// Mitsubishi GX Works2 project: 1   PLC: Q03UDV

PROGRAM P1
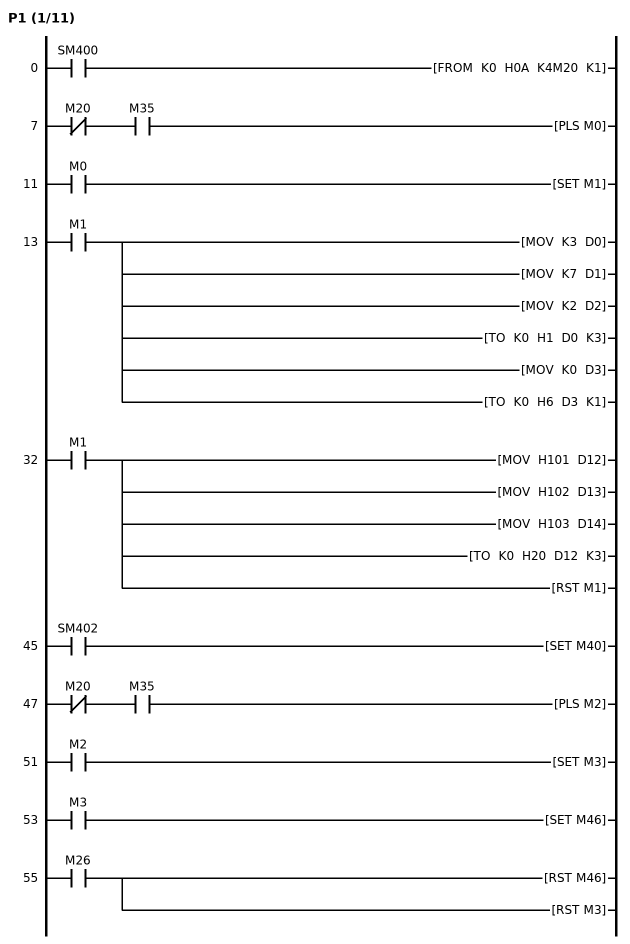
0     LD      SM400
      FROM    K0 H0A K4M20 K1
7     LDI     M20
      AND     M35
      PLS     M0
11    LD      M0
      SET     M1
13    LD      M1
      MOV     K3 D0
      MOV     K7 D1
      MOV     K2 D2
      TO      K0 H1 D0 K3
      MOV     K0 D3
      TO      K0 H6 D3 K1
32    LD      M1
      MOV     H101 D12
      MOV     H102 D13
      MOV     H103 D14
      TO      K0 H20 D12 K3
      RST     M1
45    LD      SM402
      SET     M40
47    LDI     M20
      AND     M35
      PLS     M2
51    LD      M2
      SET     M3
53    LD      M3
      SET     M46
55    LD      M26
      RST     M46
      RST     M3
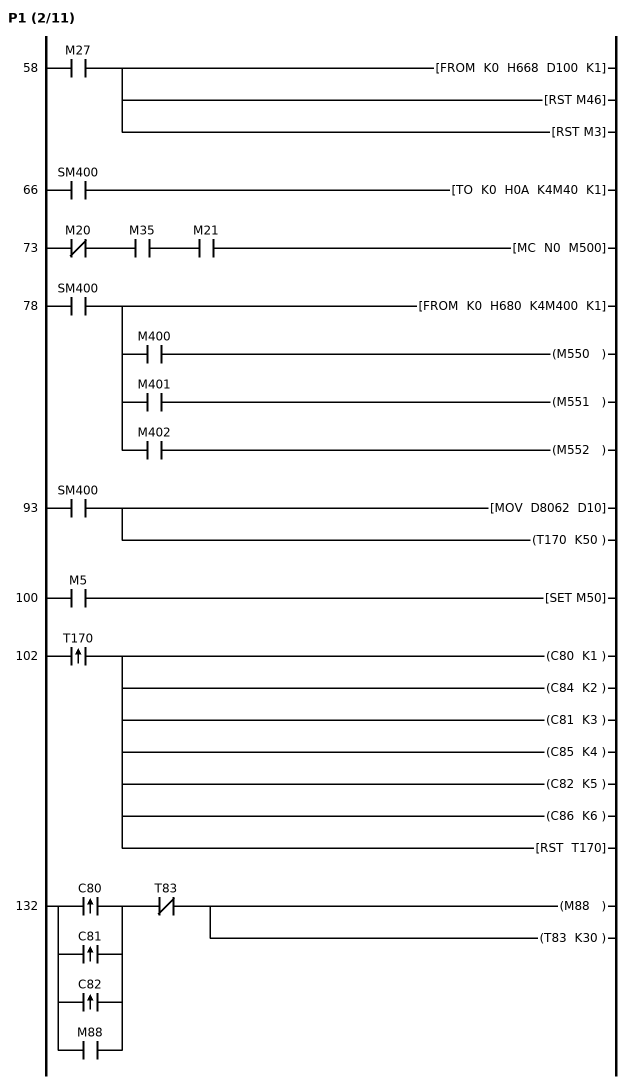
58    LD      M27
      FROM    K0 H668 D100 K1
      RST     M46
      RST     M3
66    LD      SM400
      TO      K0 H0A K4M40 K1
73    LDI     M20
      AND     M35
      AND     M21
      MC      N0 M500
78    LD      SM400
      FROM    K0 H680 K4M400 K1
      MPS
      AND     M400
      OUT     M550
      MRD
      AND     M401
      OUT     M551
      MPP
      AND     M402
      OUT     M552
93    LD      SM400
      MOV     D8062 D10
      OUT     T170 K50
100   LD      M5
      SET     M50
102   LDP     T170
      OUT     C80 K1
      OUT     C84 K2
      OUT     C81 K3
      OUT     C85 K4
      OUT     C82 K5
      OUT     C86 K6
      RST     T170
132   LDP     C80
      ORP     C81
      ORP     C82
      OR      M88
      ANI     T83
      OUT     M88
      OUT     T83 K30
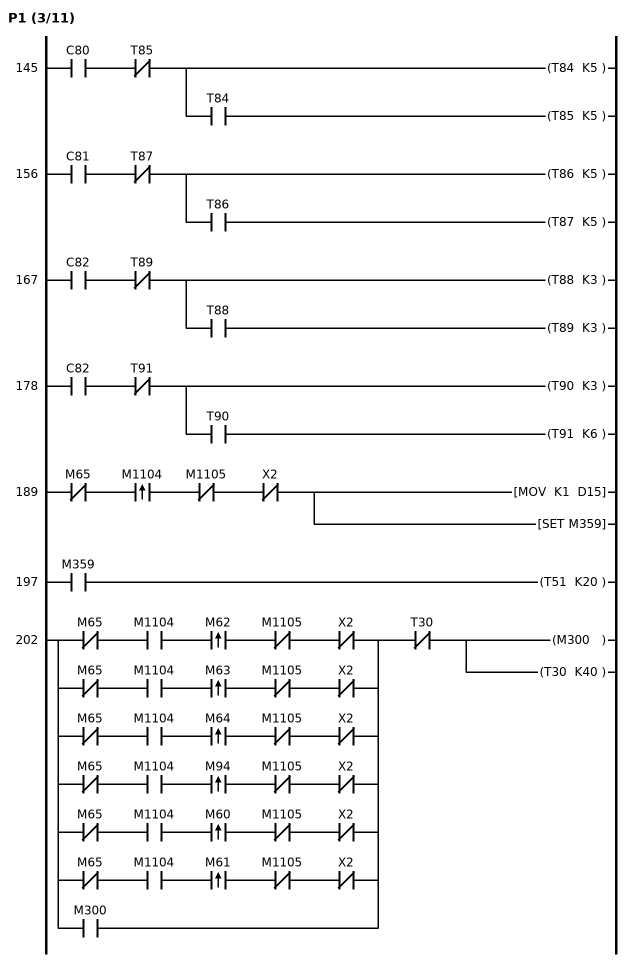
145   LD      C80
      ANI     T85
      OUT     T84 K5
      AND     T84
      OUT     T85 K5
156   LD      C81
      ANI     T87
      OUT     T86 K5
      AND     T86
      OUT     T87 K5
167   LD      C82
      ANI     T89
      OUT     T88 K3
      AND     T88
      OUT     T89 K3
178   LD      C82
      ANI     T91
      OUT     T90 K3
      AND     T90
      OUT     T91 K6
189   LDI     M65
      ANDP    M1104
      ANI     M1105
      ANI     X2
      MOV     K1 D15
      SET     M359
197   LD      M359
      OUT     T51 K20
202   LDI     M65
      AND     M1104
      ANDP    M62
      ANI     M1105
      ANI     X2
      LDI     M65
      AND     M1104
      ANDP    M63
      ANI     M1105
      ANI     X2
      ORB
      LDI     M65
      AND     M1104
      ANDP    M64
      ANI     M1105
      ANI     X2
      ORB
      LDI     M65
      AND     M1104
      ANDP    M94
      ANI     M1105
      ANI     X2
      ORB
      LDI     M65
      AND     M1104
      ANDP    M60
      ANI     M1105
      ANI     X2
      ORB
      LDI     M65
      AND     M1104
      ANDP    M61
      ANI     M1105
      ANI     X2
      ORB
      OR      M300
      ANI     T30
      OUT     M300
      OUT     T30 K40
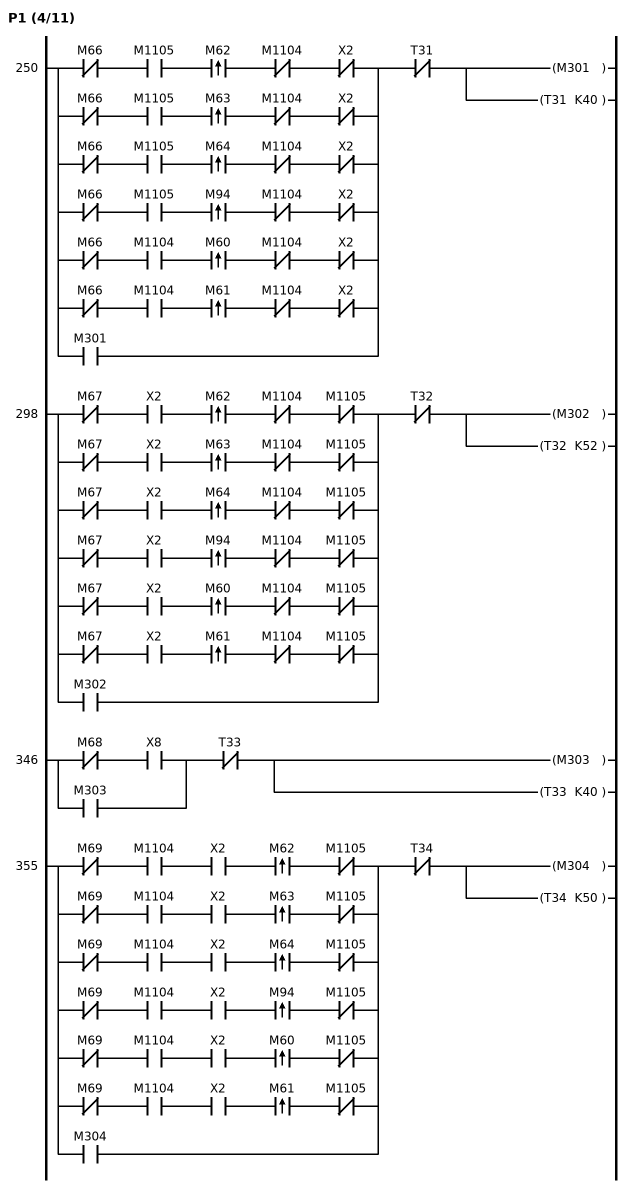
250   LDI     M66
      AND     M1105
      ANDP    M62
      ANI     M1104
      ANI     X2
      LDI     M66
      AND     M1105
      ANDP    M63
      ANI     M1104
      ANI     X2
      ORB
      LDI     M66
      AND     M1105
      ANDP    M64
      ANI     M1104
      ANI     X2
      ORB
      LDI     M66
      AND     M1105
      ANDP    M94
      ANI     M1104
      ANI     X2
      ORB
      LDI     M66
      AND     M1104
      ANDP    M60
      ANI     M1104
      ANI     X2
      ORB
      LDI     M66
      AND     M1104
      ANDP    M61
      ANI     M1104
      ANI     X2
      ORB
      OR      M301
      ANI     T31
      OUT     M301
      OUT     T31 K40
298   LDI     M67
      AND     X2
      ANDP    M62
      ANI     M1104
      ANI     M1105
      LDI     M67
      AND     X2
      ANDP    M63
      ANI     M1104
      ANI     M1105
      ORB
      LDI     M67
      AND     X2
      ANDP    M64
      ANI     M1104
      ANI     M1105
      ORB
      LDI     M67
      AND     X2
      ANDP    M94
      ANI     M1104
      ANI     M1105
      ORB
      LDI     M67
      AND     X2
      ANDP    M60
      ANI     M1104
      ANI     M1105
      ORB
      LDI     M67
      AND     X2
      ANDP    M61
      ANI     M1104
      ANI     M1105
      ORB
      OR      M302
      ANI     T32
      OUT     M302
      OUT     T32 K52
346   LDI     M68
      AND     X8
      OR      M303
      ANI     T33
      OUT     M303
      OUT     T33 K40
355   LDI     M69
      AND     M1104
      AND     X2
      ANDP    M62
      ANI     M1105
      LDI     M69
      AND     M1104
      AND     X2
      ANDP    M63
      ANI     M1105
      ORB
      LDI     M69
      AND     M1104
      AND     X2
      ANDP    M64
      ANI     M1105
      ORB
      LDI     M69
      AND     M1104
      AND     X2
      ANDP    M94
      ANI     M1105
      ORB
      LDI     M69
      AND     M1104
      AND     X2
      ANDP    M60
      ANI     M1105
      ORB
      LDI     M69
      AND     M1104
      AND     X2
      ANDP    M61
      ANI     M1105
      ORB
      OR      M304
      ANI     T34
      OUT     M304
      OUT     T34 K50
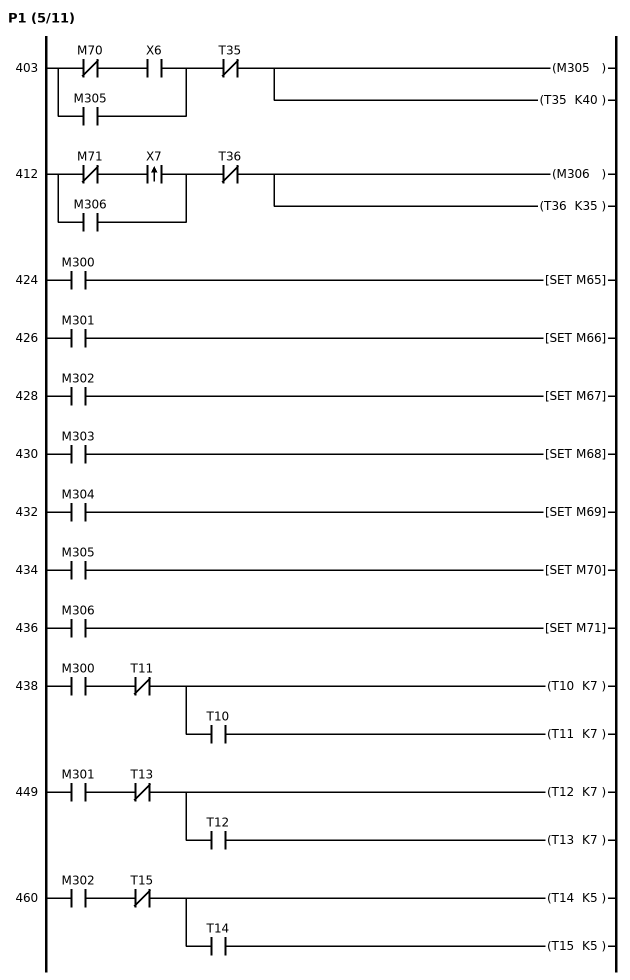
403   LDI     M70
      AND     X6
      OR      M305
      ANI     T35
      OUT     M305
      OUT     T35 K40
412   LDI     M71
      ANDP    X7
      OR      M306
      ANI     T36
      OUT     M306
      OUT     T36 K35
424   LD      M300
      SET     M65
426   LD      M301
      SET     M66
428   LD      M302
      SET     M67
430   LD      M303
      SET     M68
432   LD      M304
      SET     M69
434   LD      M305
      SET     M70
436   LD      M306
      SET     M71
438   LD      M300
      ANI     T11
      OUT     T10 K7
      AND     T10
      OUT     T11 K7
449   LD      M301
      ANI     T13
      OUT     T12 K7
      AND     T12
      OUT     T13 K7
460   LD      M302
      ANI     T15
      OUT     T14 K5
      AND     T14
      OUT     T15 K5
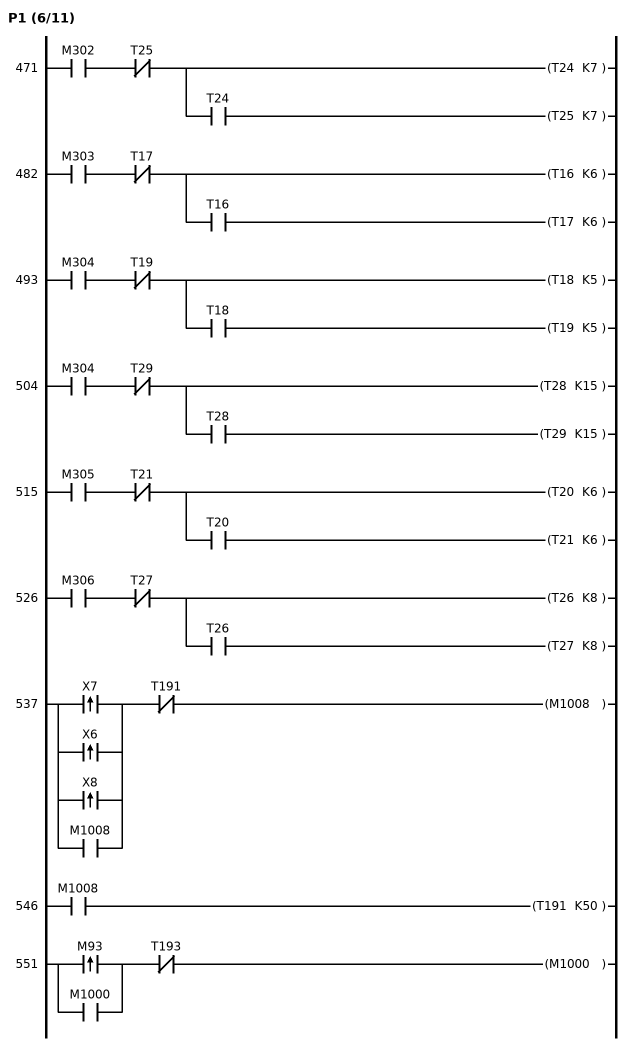
471   LD      M302
      ANI     T25
      OUT     T24 K7
      AND     T24
      OUT     T25 K7
482   LD      M303
      ANI     T17
      OUT     T16 K6
      AND     T16
      OUT     T17 K6
493   LD      M304
      ANI     T19
      OUT     T18 K5
      AND     T18
      OUT     T19 K5
504   LD      M304
      ANI     T29
      OUT     T28 K15
      AND     T28
      OUT     T29 K15
515   LD      M305
      ANI     T21
      OUT     T20 K6
      AND     T20
      OUT     T21 K6
526   LD      M306
      ANI     T27
      OUT     T26 K8
      AND     T26
      OUT     T27 K8
537   LDP     X7
      ORP     X6
      ORP     X8
      OR      M1008
      ANI     T191
      OUT     M1008
546   LD      M1008
      OUT     T191 K50
551   LDP     M93
      OR      M1000
      ANI     T193
      OUT     M1000
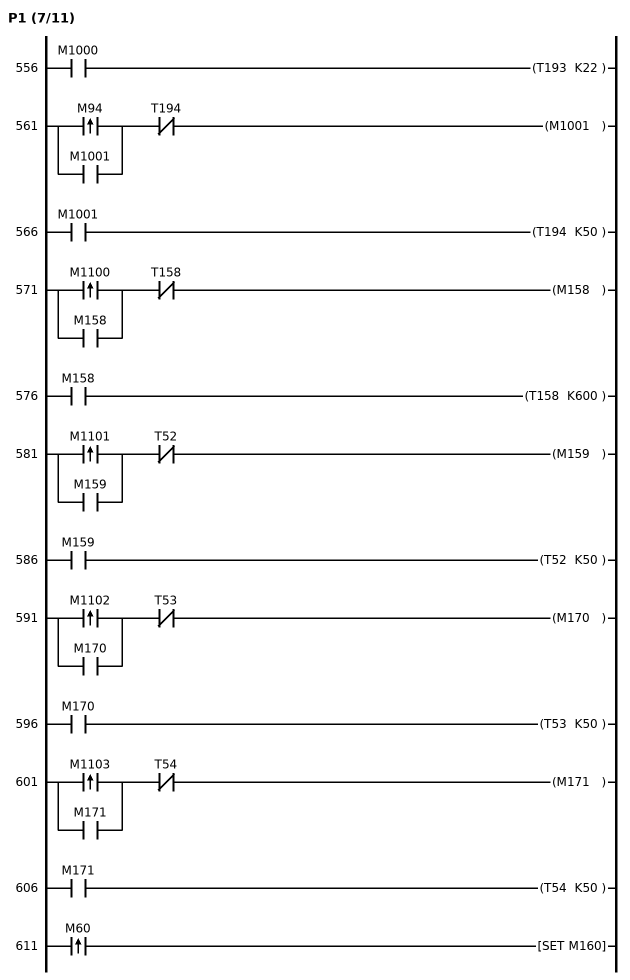
556   LD      M1000
      OUT     T193 K22
561   LDP     M94
      OR      M1001
      ANI     T194
      OUT     M1001
566   LD      M1001
      OUT     T194 K50
571   LDP     M1100
      OR      M158
      ANI     T158
      OUT     M158
576   LD      M158
      OUT     T158 K600
581   LDP     M1101
      OR      M159
      ANI     T52
      OUT     M159
586   LD      M159
      OUT     T52 K50
591   LDP     M1102
      OR      M170
      ANI     T53
      OUT     M170
596   LD      M170
      OUT     T53 K50
601   LDP     M1103
      OR      M171
      ANI     T54
      OUT     M171
606   LD      M171
      OUT     T54 K50
611   LDP     M60
      SET     M160
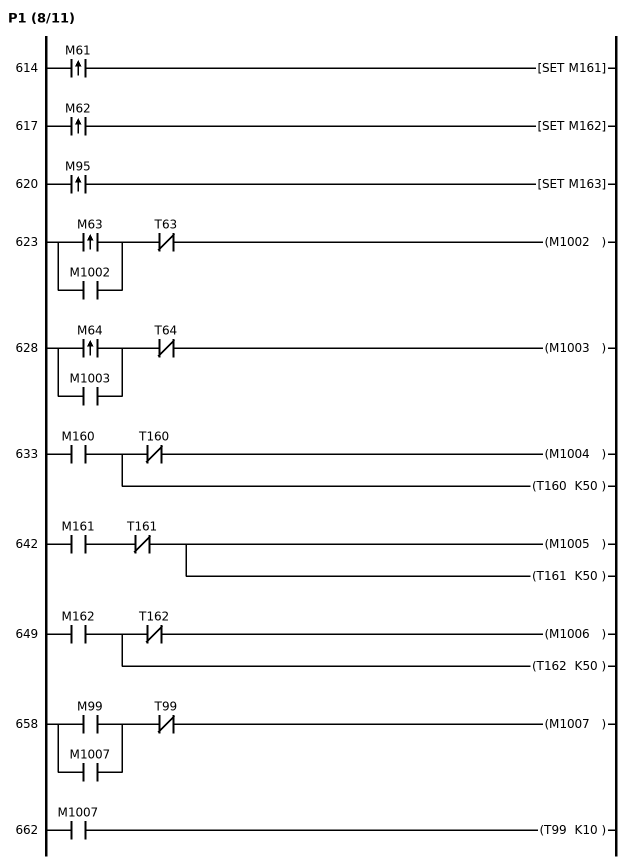
614   LDP     M61
      SET     M161
617   LDP     M62
      SET     M162
620   LDP     M95
      SET     M163
623   LDP     M63
      OR      M1002
      ANI     T63
      OUT     M1002
628   LDP     M64
      OR      M1003
      ANI     T64
      OUT     M1003
633   LD      M160
      MPS
      ANI     T160
      OUT     M1004
      MPP
      OUT     T160 K50
642   LD      M161
      ANI     T161
      OUT     M1005
      OUT     T161 K50
649   LD      M162
      MPS
      ANI     T162
      OUT     M1006
      MPP
      OUT     T162 K50
658   LD      M99
      OR      M1007
      ANI     T99
      OUT     M1007
662   LD      M1007
      OUT     T99 K10
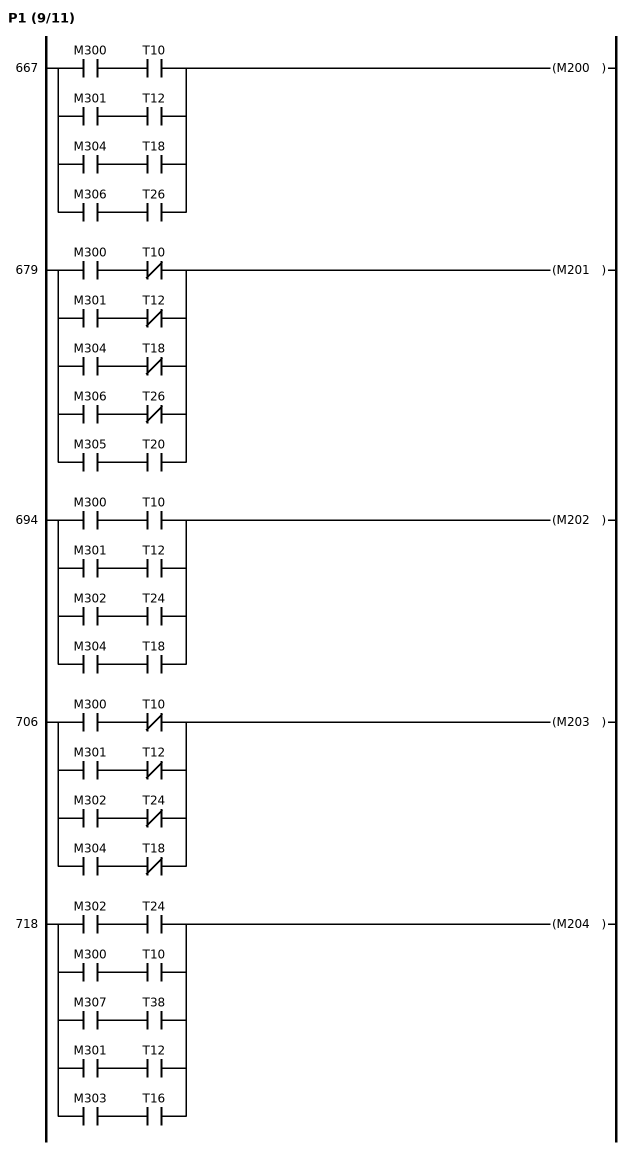
667   LD      M300
      AND     T10
      LD      M301
      AND     T12
      ORB
      LD      M304
      AND     T18
      ORB
      LD      M306
      AND     T26
      ORB
      OUT     M200
679   LD      M300
      ANI     T10
      LD      M301
      ANI     T12
      ORB
      LD      M304
      ANI     T18
      ORB
      LD      M306
      ANI     T26
      ORB
      LD      M305
      AND     T20
      ORB
      OUT     M201
694   LD      M300
      AND     T10
      LD      M301
      AND     T12
      ORB
      LD      M302
      AND     T24
      ORB
      LD      M304
      AND     T18
      ORB
      OUT     M202
706   LD      M300
      ANI     T10
      LD      M301
      ANI     T12
      ORB
      LD      M302
      ANI     T24
      ORB
      LD      M304
      ANI     T18
      ORB
      OUT     M203
718   LD      M302
      AND     T24
      LD      M300
      AND     T10
      ORB
      LD      M307
      AND     T38
      ORB
      LD      M301
      AND     T12
      ORB
      LD      M303
      AND     T16
      ORB
      OUT     M204
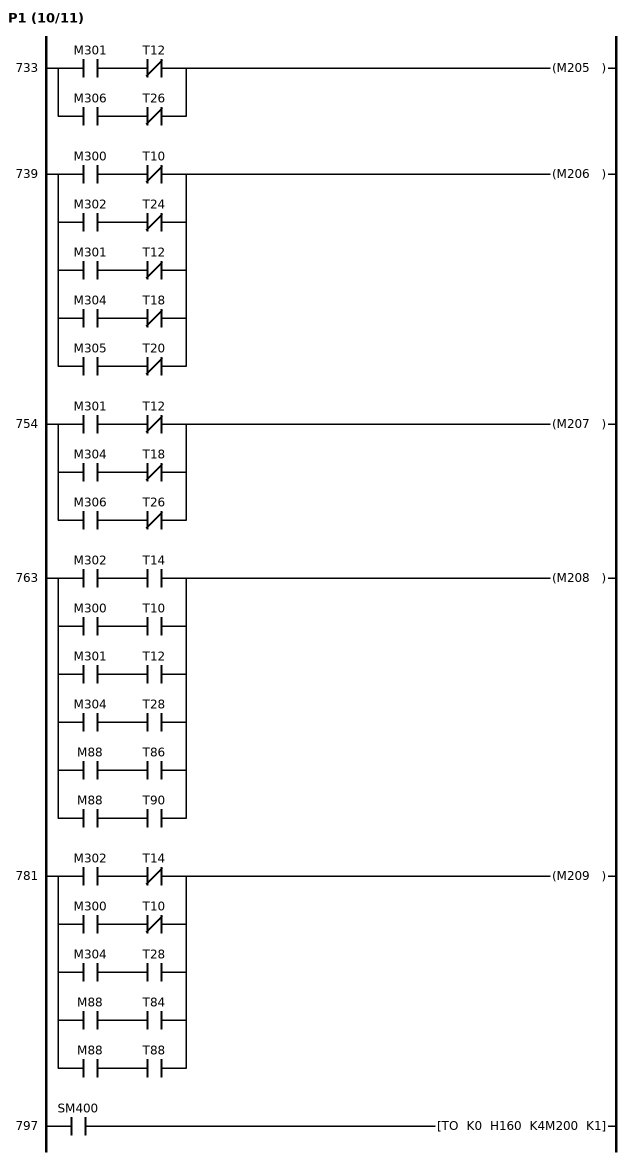
733   LD      M301
      ANI     T12
      LD      M306
      ANI     T26
      ORB
      OUT     M205
739   LD      M300
      ANI     T10
      LD      M302
      ANI     T24
      ORB
      LD      M301
      ANI     T12
      ORB
      LD      M304
      ANI     T18
      ORB
      LD      M305
      ANI     T20
      ORB
      OUT     M206
754   LD      M301
      ANI     T12
      LD      M304
      ANI     T18
      ORB
      LD      M306
      ANI     T26
      ORB
      OUT     M207
763   LD      M302
      AND     T14
      LD      M300
      AND     T10
      ORB
      LD      M301
      AND     T12
      ORB
      LD      M304
      AND     T28
      ORB
      LD      M88
      AND     T86
      ORB
      LD      M88
      AND     T90
      ORB
      OUT     M208
781   LD      M302
      ANI     T14
      LD      M300
      ANI     T10
      ORB
      LD      M304
      AND     T28
      ORB
      LD      M88
      AND     T84
      ORB
      LD      M88
      AND     T88
      ORB
      OUT     M209
797   LD      SM400
      TO      K0 H160 K4M200 K1
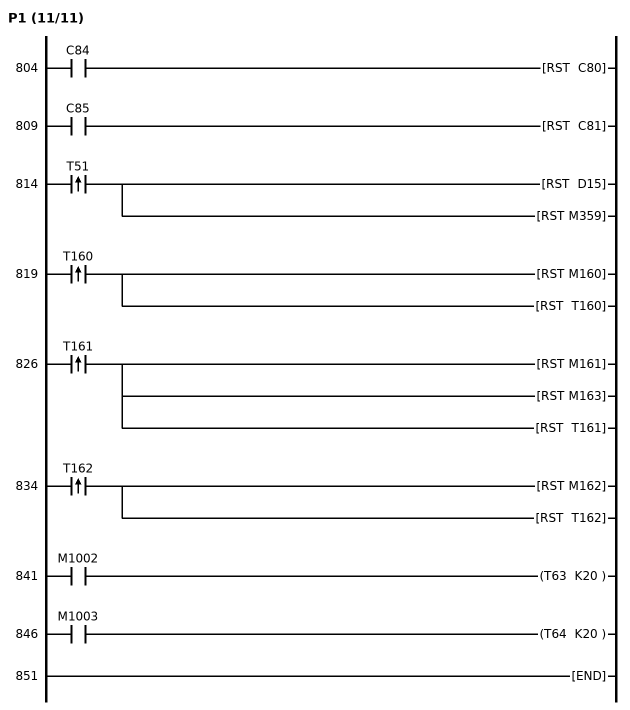
804   LD      C84
      RST     C80
809   LD      C85
      RST     C81
814   LDP     T51
      RST     D15
      RST     M359
819   LDP     T160
      RST     M160
      RST     T160
826   LDP     T161
      RST     M161
      RST     M163
      RST     T161
834   LDP     T162
      RST     M162
      RST     T162
841   LD      M1002
      OUT     T63 K20
846   LD      M1003
      OUT     T64 K20
851   END
END_PROGRAM

PROGRAM P2
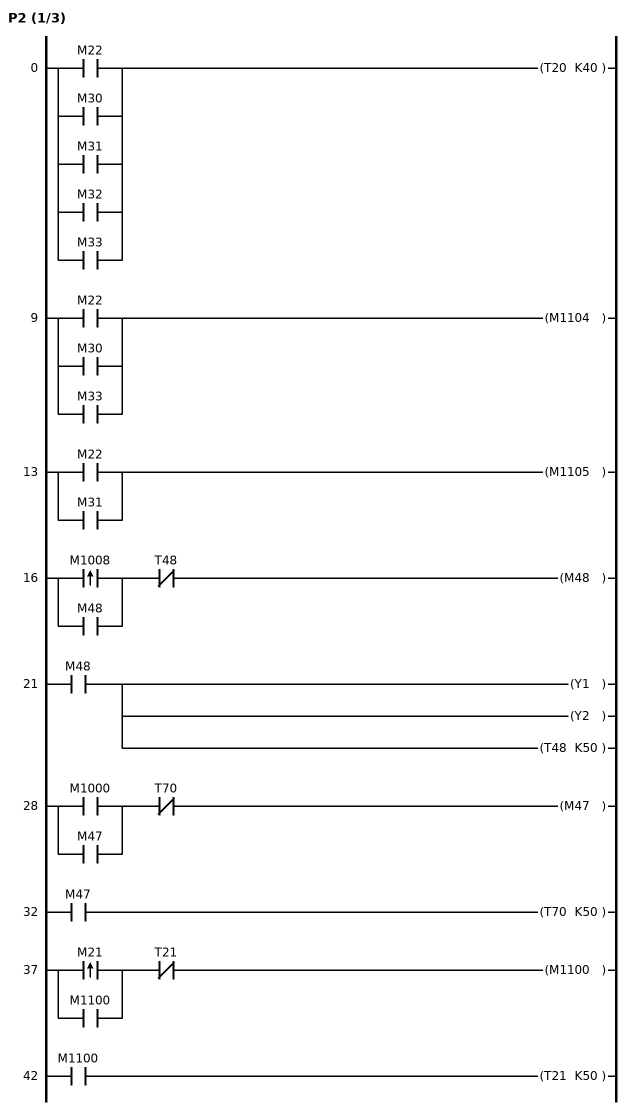
0     LD      M22
      OR      M30
      OR      M31
      OR      M32
      OR      M33
      OUT     T20 K40
9     LD      M22
      OR      M30
      OR      M33
      OUT     M1104
13    LD      M22
      OR      M31
      OUT     M1105
16    LDP     M1008
      OR      M48
      ANI     T48
      OUT     M48
21    LD      M48
      OUT     Y1
      OUT     Y2
      OUT     T48 K50
28    LD      M1000
      OR      M47
      ANI     T70
      OUT     M47
32    LD      M47
      OUT     T70 K50
37    LDP     M21
      OR      M1100
      ANI     T21
      OUT     M1100
42    LD      M1100
      OUT     T21 K50
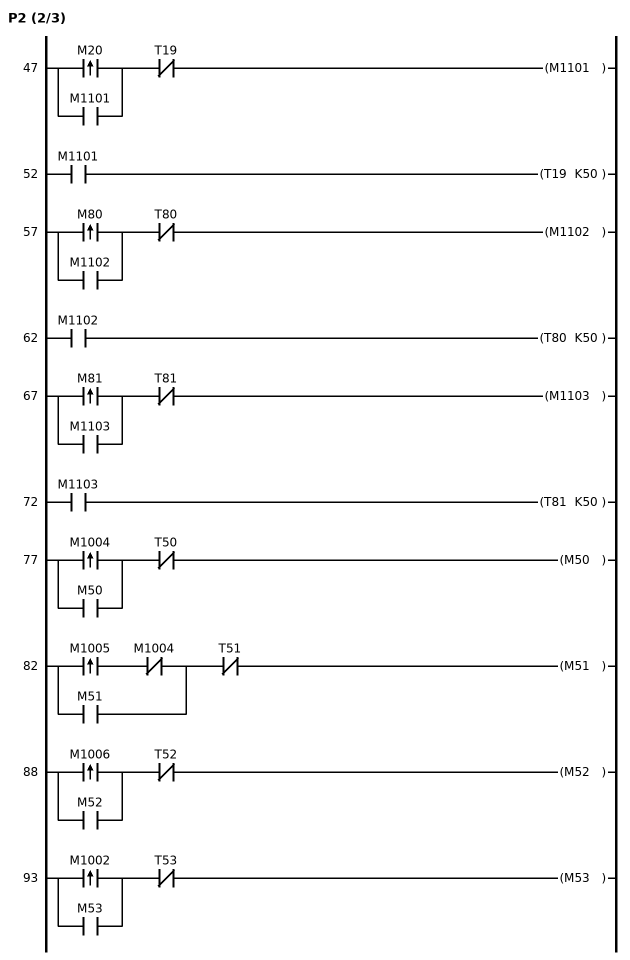
47    LDP     M20
      OR      M1101
      ANI     T19
      OUT     M1101
52    LD      M1101
      OUT     T19 K50
57    LDP     M80
      OR      M1102
      ANI     T80
      OUT     M1102
62    LD      M1102
      OUT     T80 K50
67    LDP     M81
      OR      M1103
      ANI     T81
      OUT     M1103
72    LD      M1103
      OUT     T81 K50
77    LDP     M1004
      OR      M50
      ANI     T50
      OUT     M50
82    LDP     M1005
      ANI     M1004
      OR      M51
      ANI     T51
      OUT     M51
88    LDP     M1006
      OR      M52
      ANI     T52
      OUT     M52
93    LDP     M1002
      OR      M53
      ANI     T53
      OUT     M53
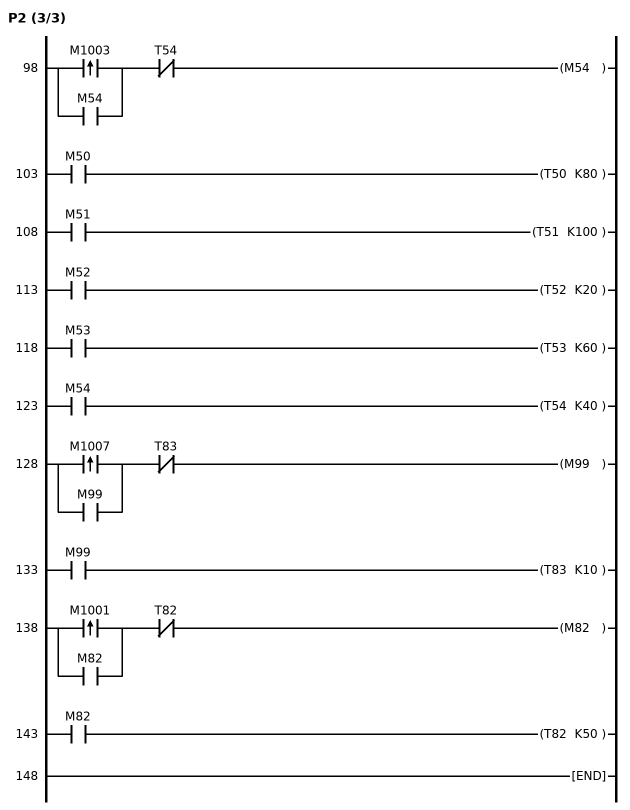
98    LDP     M1003
      OR      M54
      ANI     T54
      OUT     M54
103   LD      M50
      OUT     T50 K80
108   LD      M51
      OUT     T51 K100
113   LD      M52
      OUT     T52 K20
118   LD      M53
      OUT     T53 K60
123   LD      M54
      OUT     T54 K40
128   LDP     M1007
      OR      M99
      ANI     T83
      OUT     M99
133   LD      M99
      OUT     T83 K10
138   LDP     M1001
      OR      M82
      ANI     T82
      OUT     M82
143   LD      M82
      OUT     T82 K50
148   END
END_PROGRAM
